{attribute 'no_explicit_call' := 'do not call this function block directly'} 
// The wrapper around Tc2_Standard.TON
FUNCTION_BLOCK FINAL SequentialTaskExecutor EXTENDS Core.AbortableProcess
VAR
	{attribute 'OPC.UA.DA' := '0'}
	_ClassName : STRING := __POUNAME();

	{attribute 'OPC.UA.DA' := '0'}
	_Tasks : Collections.List;
	
	{attribute 'OPC.UA.DA' := '0'}
	_ContinueOnError : BOOL;
END_VAR

{attribute 'monitoring' := 'call'}
PROPERTY ClassName : STRING
GET
ClassName := _ClassName;
END_GET
END_PROPERTY

{attribute 'monitoring' := 'call'}
PROPERTY ContinueOnError : BOOL
GET
ContinueOnError := _ContinueOnError;
END_GET
END_PROPERTY

{attribute 'monitoring' := 'call'}
PROPERTY CurrentTask : IAbortableTask
GET
IF _Tasks.Count > 0 THEN
	__QUERYINTERFACE(_Tasks.Get(0).AsObject(), CurrentTask);
END_IF
END_GET
END_PROPERTY

{attribute 'monitoring' := 'call'}
{attribute 'OPC.UA.DA.Property' := '1'}
{attribute 'OPC.UA.DA.Access' := '1'}
PROPERTY Name : WSTRING
GET
Name := TO_WSTRING(ClassName);
END_GET
END_PROPERTY

METHOD PROTECTED OnAbort 
VAR_INPUT
	start : BOOL;
END_VAR
VAR_OUTPUT
	done : BOOL;
END_VAR
VAR
	task : Core.IAbortableTask;

	exceptionCode : __SYSTEM.ExceptionCode;
END_VAR
IF _Tasks.Count < 1 THEN
	done := TRUE;
	RETURN;
END_IF

task := CurrentTask;

__TRY
	IF start THEN
		task.Abort();
	ELSE
		task.Execute();
	END_IF
	
	IF NOT task.Busy THEN
		_Tasks.RemoveAt(0);
		done := TRUE;
	END_IF
__CATCH(exceptionCode)
	IF _Tasks.Count > 0 THEN
		_Tasks.RemoveAt(0);
	END_IF
	
	IF ContinueOnError THEN
		done := TRUE;
	ELSE
		Core.ExceptionManager.Throw(Core.ExceptionManager.GetLastException(exceptionCode));
	END_IF	
__ENDTRY
END_METHOD

METHOD PROTECTED OnRun 
VAR_INPUT
	start : BOOL;
END_VAR
VAR
	task : Core.IAbortableTask;

	exceptionCode : __SYSTEM.ExceptionCode;
END_VAR
IF _Tasks.Count < 1 THEN
	RETURN;
END_IF

task := CurrentTask;

__TRY
	IF start OR_ELSE NOT task.Busy THEN
		task.Start();
	ELSE
		task.Execute();
	END_IF
	
	IF NOT task.Busy THEN
		_Tasks.RemoveAt(0);
	END_IF
__CATCH(exceptionCode)
	IF _Tasks.Count > 0 THEN
		_Tasks.RemoveAt(0);
	END_IF
	
	IF NOT ContinueOnError THEN
		Core.ExceptionManager.Throw(Core.ExceptionManager.GetLastException(exceptionCode));
	END_IF
__ENDTRY
END_METHOD

METHOD ScheduleTask
VAR_INPUT
	task : Core.IAbortableTask;
	releseAfterHandling : BOOL;
END_VAR
_Tasks.AppendGeneric(Core.GenericValueFactory.FromParts(DATA_TYPE.TYPE_OBJECT, task.Address, task.Size, releseAfterHandling));
END_METHOD

{attribute 'monitoring' := 'call'}
PROPERTY Size : ULINT
GET
Size := XSIZEOF(THIS^);
END_GET
END_PROPERTY

END_FUNCTION_BLOCK

(* stored: Version 1.1.0.1
   POU SequentialTaskExecutor: Id {5f2d9604-eb7b-45e3-84bc-b901136bbe0b}, SpecialFunc None
   Folder Overriden: Id {1b1c5863-9f32-4a15-87e0-d0e2df5c3f78}
   Property ClassName: Id {ba95610f-5219-47c9-8c57-311d9e60e72f}
   Get Get: Id {013b3af7-a06d-4fbf-a280-1144598a7235}
   Property ContinueOnError: Id {46940bfd-6bf9-4e6a-8051-ecad3e387b69}
   Get Get: Id {3f04ff4a-f44d-4d07-bfe1-9565fe1e2fca}
   Property CurrentTask: Id {c0d02002-6e75-4b84-a496-ad82ebf3d647}
   Get Get: Id {28df5953-696c-4fdc-b8d7-69723340165e}
   Property Name: Id {877e85fd-25b7-42c3-b3a5-1da824b3a170}
   Get Get: Id {5d3ae67f-607f-4e82-af9f-014cbc19ee29}
   Method OnAbort: Id {3a5ab894-6d0b-4ec0-b72f-2b4254f65f95}
   Method OnRun: Id {2c7c0cfd-db41-4ccf-92fc-38a7fc6a065c}
   Method ScheduleTask: Id {25e72a79-e8be-4012-84f7-5da4f4f9148b}
   Property Size: Id {b289e881-1f3e-4abc-9a70-4494d509b71b}
   Get Get: Id {40179bbc-4746-4890-bbcf-233fb2a96bdf} *)
